// TIA Portal V20 export
DATA_BLOCK "CallEquipment_DB"   // DB93
{ DB_Accessible_From_OPC_UA := 'FALSE' }
// stored: AssignedProDiagFB Unit1.Em6.ProDiag, DBAccessibleFromOPCUA false, DBAccessibleFromWebserver false, InstanceOfName Unit1.Em6.CallEquipment, InstanceOfType FB, Namespace Unit1.Em6
"Unit1.Em6.CallEquipment"
   // VAR_INPUT
   //    ZoneOperationEnable { ExternalWritable := 'False'} : "LWONIK_typeSafetyZoneManualOperation";
   //    unitEnableControlInterfaces { ExternalWritable := 'False'} : "LAF_typeEnableControlInterfaces";
   //    commandExcute { ExternalWritable := 'False'} : Bool;
   // END_VAR
   // VAR_IN_OUT
   //    unitStatus : "LAF_typeUnitStatus";
   //    emFeedback : "LUC_typeEmFeedback";
   //    unitAlarmDB : "LAF_typeAlarms";
   // END_VAR
   // VAR
   //    instSequenceVisionUnit { ExternalWritable := 'False'} : "Unit1.Em6.Sequence_1_VisionUnit";
   //    instSequenceVisionController { ExternalWritable := 'False'} : "Unit1.Em6.Sequence_2_VisionController";
   //    instSequenceQrRead { ExternalWritable := 'False'} : "Unit1.Em6.Sequence_3_QrRead";
   //    instVisionUnitInitializedJob1 { ExternalWritable := 'False'} : "LAF_SelectJob";
   //    instVisionUnitVisionPosJob2 { ExternalWritable := 'False'} : "LAF_SelectJob";
   //    instVisionUnitHomePosJob3 { ExternalWritable := 'False'} : "LAF_SelectJob";
   //    instVisionFullAutoJob10 { ExternalWritable := 'False'} : "LAF_SelectJob";
   //    instVisionControllerInitializedJob1 { ExternalWritable := 'False'} : "LAF_SelectJob";
   //    instVisionControllerInspectionJob2 { ExternalWritable := 'False'} : "LAF_SelectJob";
   //    instQrReaderInitializedJob1 { ExternalWritable := 'False'} : "LAF_SelectJob";
   //    instQrReaderQrReadJob2 { ExternalWritable := 'False'} : "LAF_SelectJob";
   //    instCmVisionAxisZ { ExternalWritable := 'False'} : "LBC_Axis64Pos_TecPlcCn";
   //    instCmVisionPusherSupportUpDown { ExternalWritable := 'False'} : "LBC_TwoWayActuatorCn";
   //    instCmVisionTriggerSensor { ExternalWritable := 'False'} : "LBC_DigitalSignalCn";
   //    instCmQrReader { ExternalWritable := 'False'} : "LER_QRread_SRX300";
   //    instCmQrReadHandy { ExternalWritable := 'False'} : "LER_QRread_DM8700";
   //    instVision_XGX2000 { ExternalWritable := 'False'} : "LER_Vision_XGX2000";
   //    instVision_XGX2000_Conversion { ExternalWritable := 'False'} : "LER_Vision_XGX2000_Conversion";
   //    instVisionAxisZControlInterlockSummary { ExternalWritable := 'False'} : "LER_Axis64Pos_InterlockSummary";
   //    instServoTorqueCal_DR9 { ExternalWritable := 'False'} : "LER_ServoTorqueCal";
   //    instLDrv701ControlVisionAxisZ { ExternalWritable := 'False'} : "LDrvSafe_SinaTlg701Control";
   //    instLDrv701StatusVisionAxisZ { ExternalWritable := 'False'} : "LDrvSafe_SinaTlg701Status";
   //    statUnitStatus { ExternalWritable := 'False'} : "LAF_typeUnitStatus";
   //    statAllBrakeTest { ExternalWritable := 'False'} : "LER_typeBrakeTestUnitCommands";
   //    instManageAlarms { ExternalWritable := 'False'} : "LAF_ManageAlarms";
   //    instEventsPFE { S7_SetPoint := 'True'} : "Unit1.Em6.EventsPFE";
   //    statPulse { ExternalWritable := 'False'} : Array[0..99] of Bool;
   //    statTonTimer { ExternalWritable := 'False'} : Array[0..99] of TON_TIME;
   //    statTofTimer { ExternalWritable := 'False'} : Array[0..99] of TOF_TIME;
   //    statEnableManualCmds { ExternalWritable := 'False'} : Bool;
   //    statGaugeCheck { ExternalWritable := 'False'} : Struct
   //       Type1Complete : Bool;
   //       Type3Compete : Bool;
   //    END_STRUCT;
   //    statSafeStateCheck { ExternalWritable := 'False'} : Struct
   //       VisionUnit : Bool;
   //       VisionController : Bool;
   //       VisionQrReader : Bool;
   //    END_STRUCT;
   //    statBobinID : String[32];
   //    citi_Ptrig : Array[0..20] of Bool;
   //    citiTon : Array[0..20] of TON_TIME;
   //    citi : Time;
   //    citiTest : Array[0..20] of Bool;
   //    statDataIncrease : Int;
   // END_VAR
BEGIN
END_DATA_BLOCK
